(* Schneider Machine Expert - Basic project tank_level_v5_TM221CE16T, file version 3.0.0.0 *)
(* ProjectInformations: Name=Tank Level Control v5 with TM3AI4/G *)

HARDWARE
  Cpu 0: TM221CE16T
  ModuleExtensionObject 0: TM3AI4/G
  EthernetConfiguration: NetworkName=M221, IpAllocationMode=ByDhcp, IpAddress=192.168.1.10, SubnetMask=255.255.255.0
  SerialLineConfiguration: Baud=Baud19200, Parity=ParityEven, DataBits=DataBits8, StopBits=StopBits1, PhysicalMedium=PhysicalMediumRs485, TransmissionMode=TransmissionModeModbusRtu, SlaveId=1, Addressing=SlaveAddressing
  MastTask: UsePeriodScanMode=false, PeriodScan=100
  FastTask: Period=255
  CpuBehavior: StartingMode=StartAsPreviousState, AutoSaveRamOnEeprom=true, WatchdogPeriod=250

SYMBOLS  (address, symbol, comment, settings)
  %M0       TANK_FULL  "Tank full flag from ultrasonic sensor"
  %M1       TANK_EMPTY  "Tank empty flag from ultrasonic sensor"
  %MW0      LEVEL_RAW  "Raw analog value from ultrasonic sensor for HMI"
  %Q0.0     INLET_VLV  "Inlet valve solenoid"
  %Q0.1     OUTLET_VLV  "Outlet valve solenoid"
  %IW1.0    LEVEL_AIN  "Ultrasonic level transmitter 4-20mA"  [Type=Type_4_20mA, Scope=Scope_Normal, Minimum=0, Maximum=10000]

POU Tank Level Control
  (* SectionNumber=0 *)

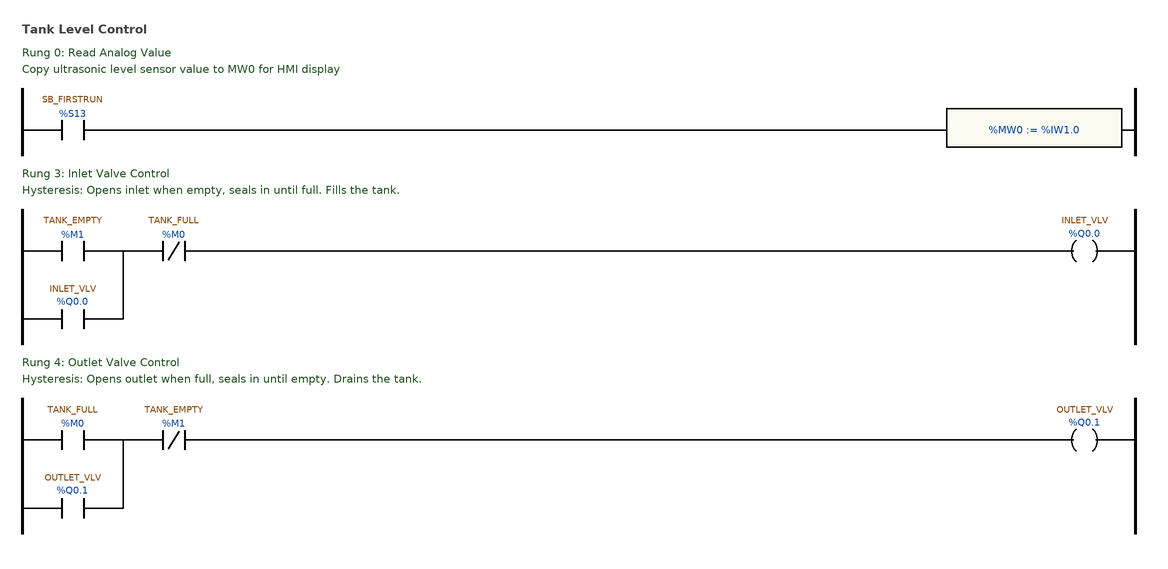

// Rung 0: Read Analog Value
// Copy ultrasonic level sensor value to MW0 for HMI display
  LD %S13
  [ %MW0 := %IW1.0 ]      (* LEVEL_RAW, LEVEL_AIN *)
  // as ST:
  //   IF %S13 THEN LEVEL_RAW := LEVEL_AIN; END_IF;

// Rung 1: Tank Full Detection
// Ultrasonic sensor: low value means tank full. Set flag when level below 1800.
  LD [%IW1.0<1800]        (* LEVEL_AIN *)
  ST %M0                  (* TANK_FULL *)
  // as ST:
  //   TANK_FULL := LEVEL_AIN<1800;
  (* the ladder stored for this rung does not match its IL; not drawn *)

// Rung 2: Tank Empty Detection
// Ultrasonic sensor: high value means tank empty. Set flag when level above 4800.
  LD [%IW1.0>4800]        (* LEVEL_AIN *)
  ST %M1                  (* TANK_EMPTY *)
  // as ST:
  //   TANK_EMPTY := LEVEL_AIN>4800;
  (* the ladder stored for this rung does not match its IL; not drawn *)

// Rung 3: Inlet Valve Control
// Hysteresis: Opens inlet when empty, seals in until full. Fills the tank.
  LD %M1                  (* TANK_EMPTY *)
  OR %Q0.0                (* INLET_VLV *)
  ANDN %M0                (* TANK_FULL *)
  ST %Q0.0                (* INLET_VLV *)
  // as ST:
  //   INLET_VLV := (TANK_EMPTY OR INLET_VLV) AND NOT TANK_FULL;

// Rung 4: Outlet Valve Control
// Hysteresis: Opens outlet when full, seals in until empty. Drains the tank.
  LD %M0                  (* TANK_FULL *)
  OR %Q0.1                (* OUTLET_VLV *)
  ANDN %M1                (* TANK_EMPTY *)
  ST %Q0.1                (* OUTLET_VLV *)
  // as ST:
  //   OUTLET_VLV := (TANK_FULL OR OUTLET_VLV) AND NOT TANK_EMPTY;
